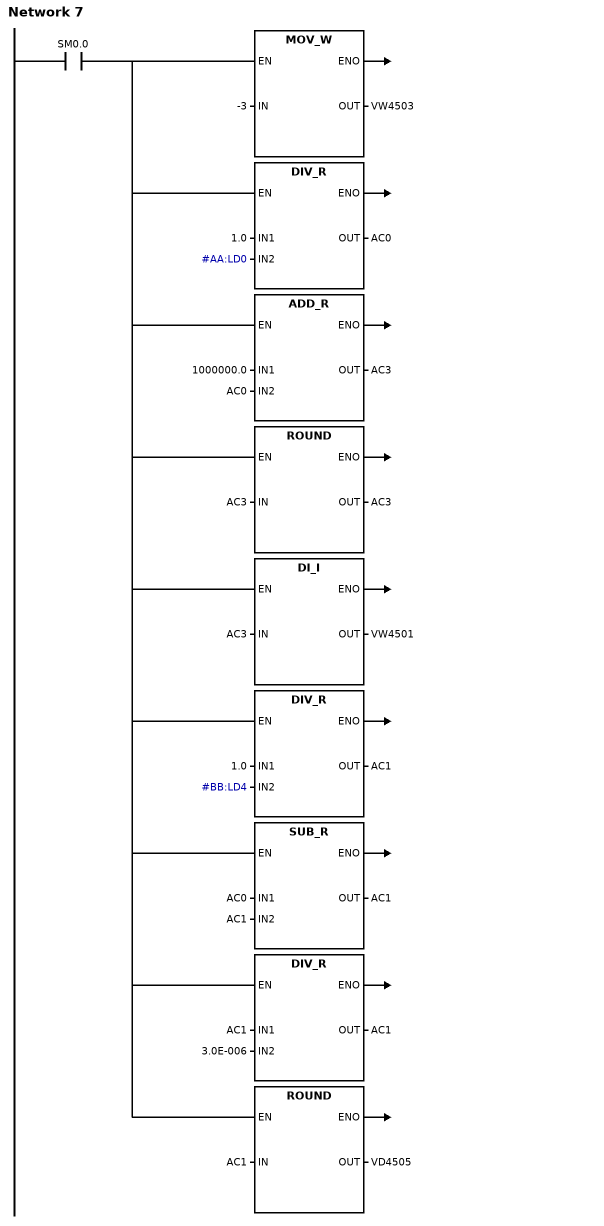
[picture p24: SBR5 networks 7-7]
Network 7
LD     SM0.0
MOVW   -3, VW4503
MOVR   1.0, AC0
/R     #AA:LD0, AC0
MOVR   1000000.0, AC3
+R     AC0, AC3
ROUND  AC3, AC3
DTI    AC3, VW4501
MOVR   1.0, AC1
/R     #BB:LD4, AC1
*R     -1.0, AC1
+R     AC0, AC1
/R     3.0E-006, AC1
ROUND  AC1, VD4505
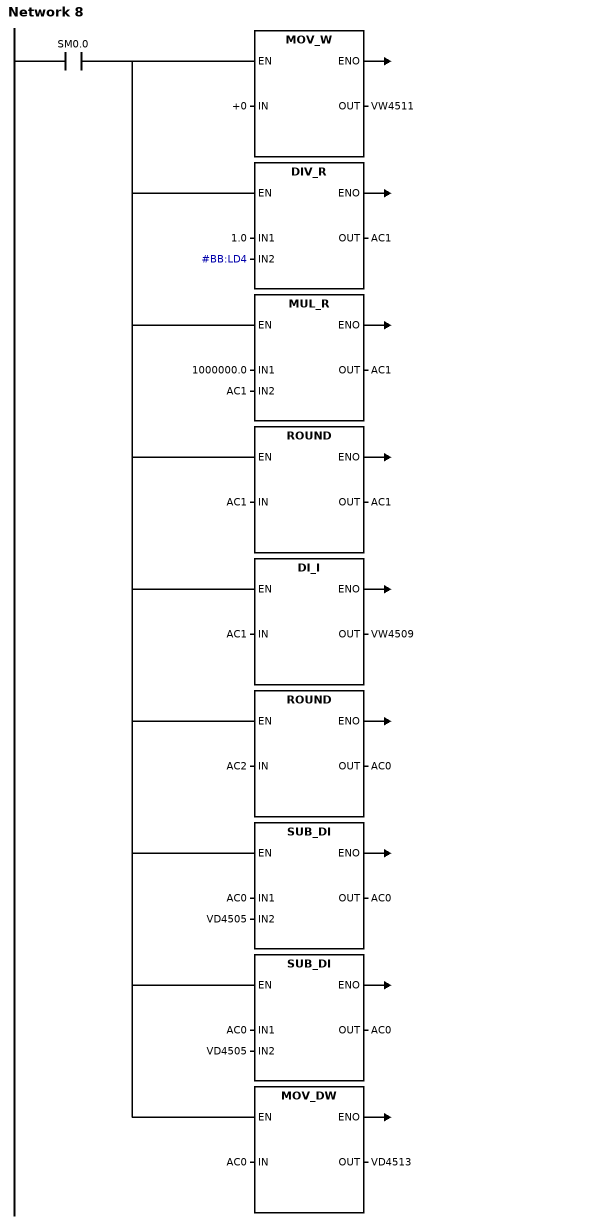
Network 8
LD     SM0.0
MOVW   +0, VW4511
MOVR   1.0, AC1
/R     #BB:LD4, AC1
*R     1000000.0, AC1
ROUND  AC1, AC1
DTI    AC1, VW4509
ROUND  AC2, AC0
-D     VD4505, AC0
-D     VD4505, AC0
MOVD   AC0, VD4513
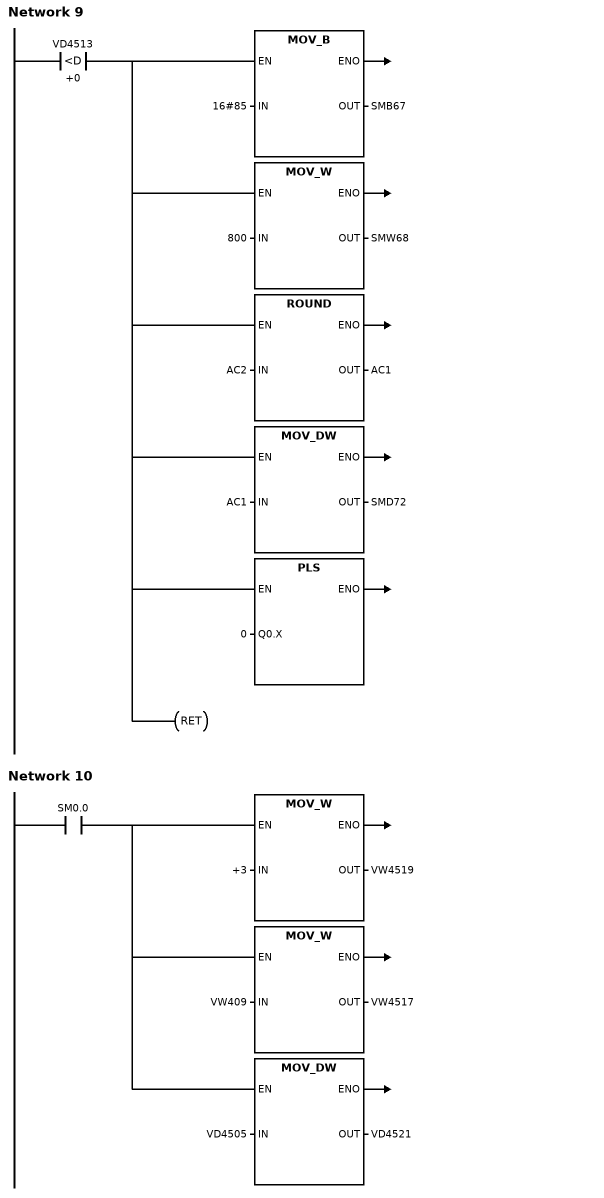
Network 9
LDD<   VD4513, +0
MOVB   16#85, SMB67
MOVW   800, SMW68
ROUND  AC2, AC1
MOVD   AC1, SMD72
PLS    0
CRET
Network 10
LD     SM0.0
MOVW   +3, VW4519
MOVW   VW409, VW4517
MOVD   VD4505, VD4521
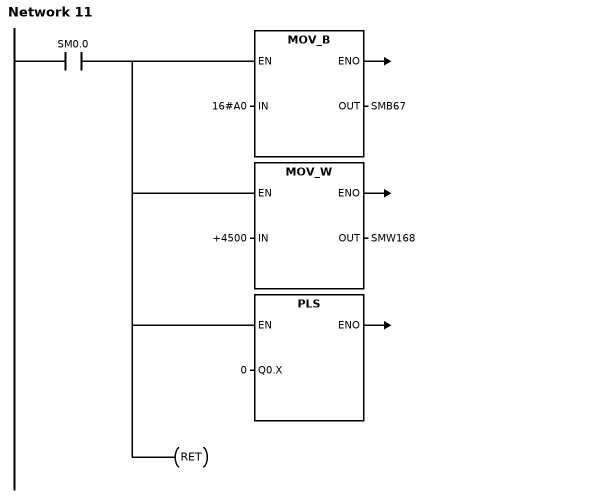
Network 11
LD     SM0.0
MOVB   16#A0, SMB67
MOVW   +4500, SMW168
PLS    0
CRET
END_SUBROUTINE_BLOCK

SUBROUTINE_BLOCK stop_ch0:SBR6
TITLE=stop_ch0
BEGIN
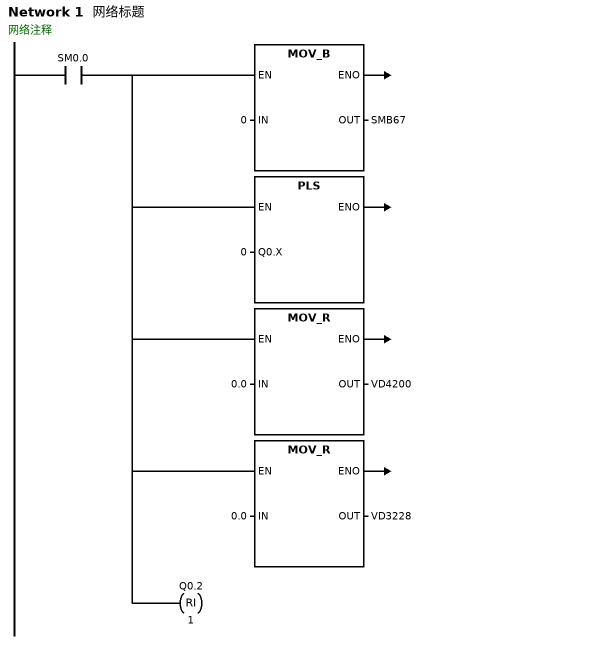
Network 1 // 网络标题
// 网络注释
LD     SM0.0
MOVB   0, SMB67
PLS    0
MOVR   0.0, VD4200
MOVR   0.0, VD3228
RI     Q0.2, 1
END_SUBROUTINE_BLOCK

SUBROUTINE_BLOCK pls_ch1:SBR7
TITLE=子程序7  //脉冲发生器2的控制程序
VAR_INPUT
AA:REAL;	// LD0 
BB:REAL;	// LD4 
CC:REAL;	// LD8 
END_VAR
BEGIN
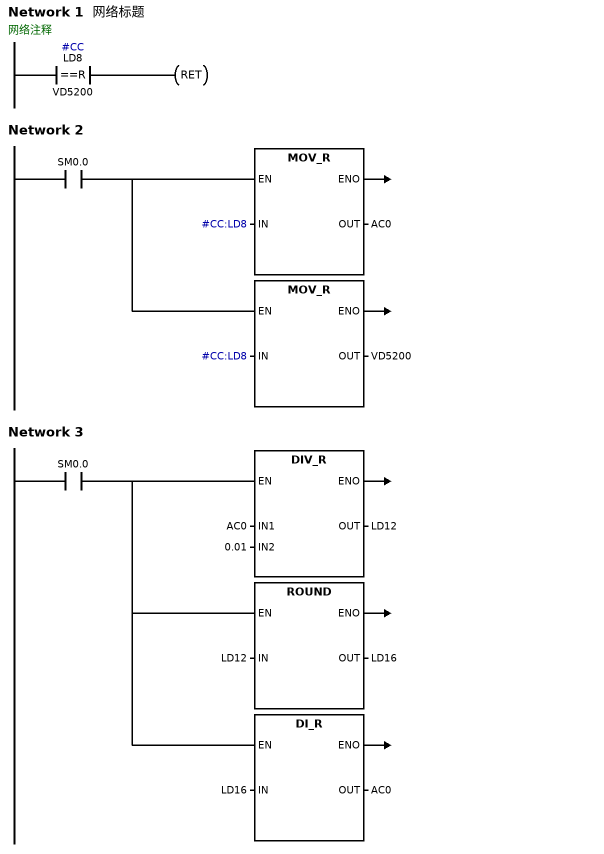
Network 1 // 网络标题
// 网络注释
LDR=   #CC:LD8, VD5200
CRET
Network 2
LD     SM0.0
MOVR   #CC:LD8, AC0
MOVR   #CC:LD8, VD5200
Network 3
LD     SM0.0
MOVR   AC0, LD12
/R     0.01, LD12
ROUND  LD12, LD16
DTR    LD16, AC0
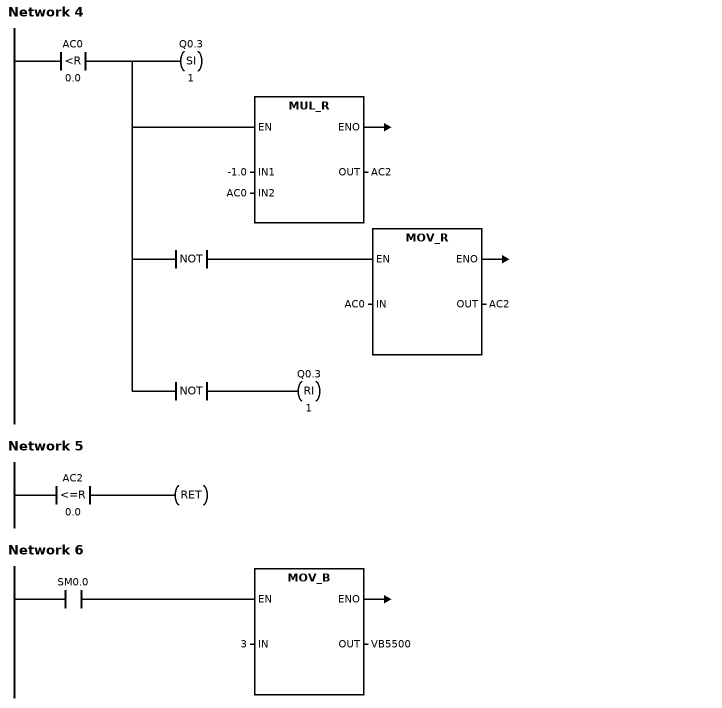
Network 4
LDR<   AC0, 0.0
LPS
SI     Q0.3, 1
MOVR   -1.0, AC2
*R     AC0, AC2
NOT
MOVR   AC0, AC2
LPP
NOT
RI     Q0.3, 1
Network 5
LDR<=  AC2, 0.0
CRET
Network 6
LD     SM0.0
MOVB   3, VB5500
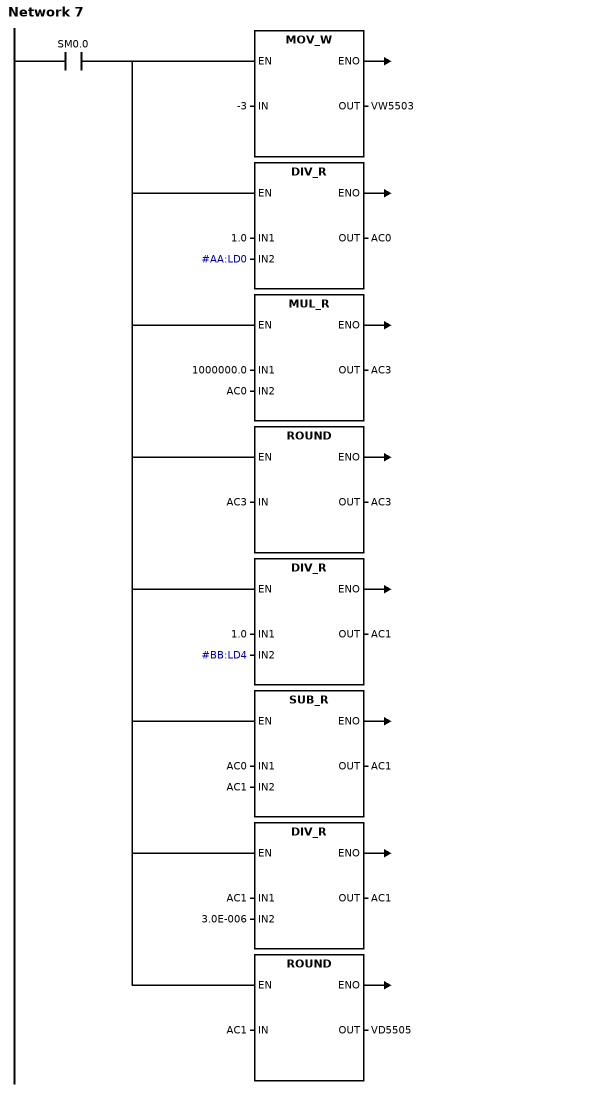
Network 7
LD     SM0.0
MOVW   -3, VW5503
MOVR   1.0, AC0
/R     #AA:LD0, AC0
MOVR   1000000.0, AC3
*R     AC0, AC3
ROUND  AC3, AC3
MOVR   1.0, AC1
/R     #BB:LD4, AC1
*R     -1.0, AC1
+R     AC0, AC1
/R     3.0E-006, AC1
ROUND  AC1, VD5505
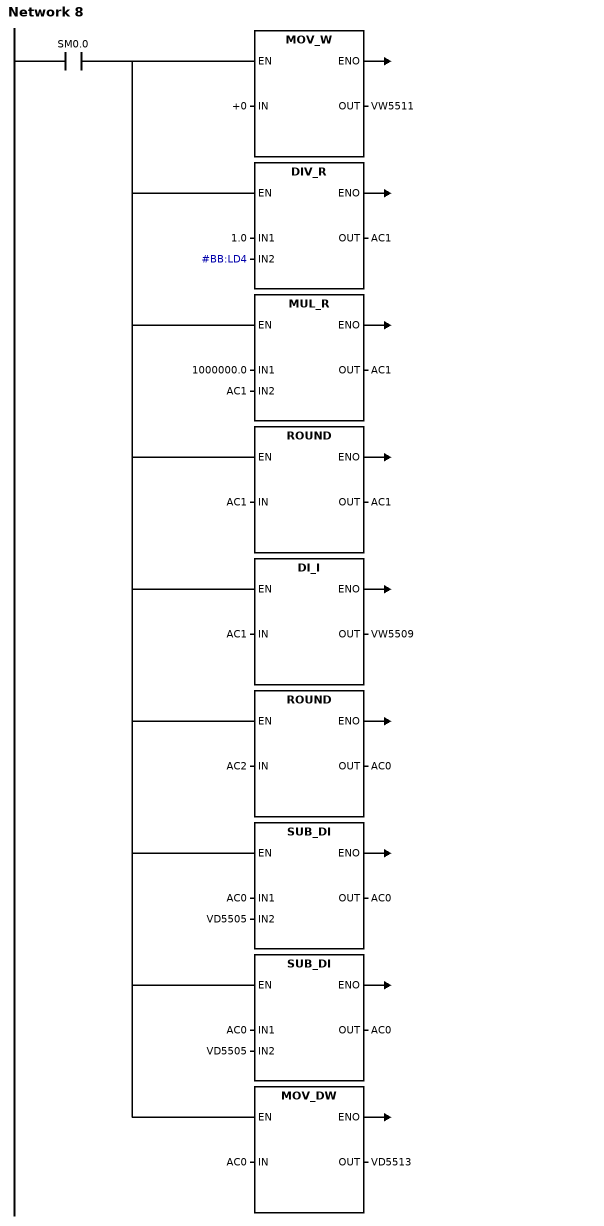
Network 8
LD     SM0.0
MOVW   +0, VW5511
MOVR   1.0, AC1
/R     #BB:LD4, AC1
*R     1000000.0, AC1
ROUND  AC1, AC1
DTI    AC1, VW5509
ROUND  AC2, AC0
-D     VD5505, AC0
-D     VD5505, AC0
MOVD   AC0, VD5513
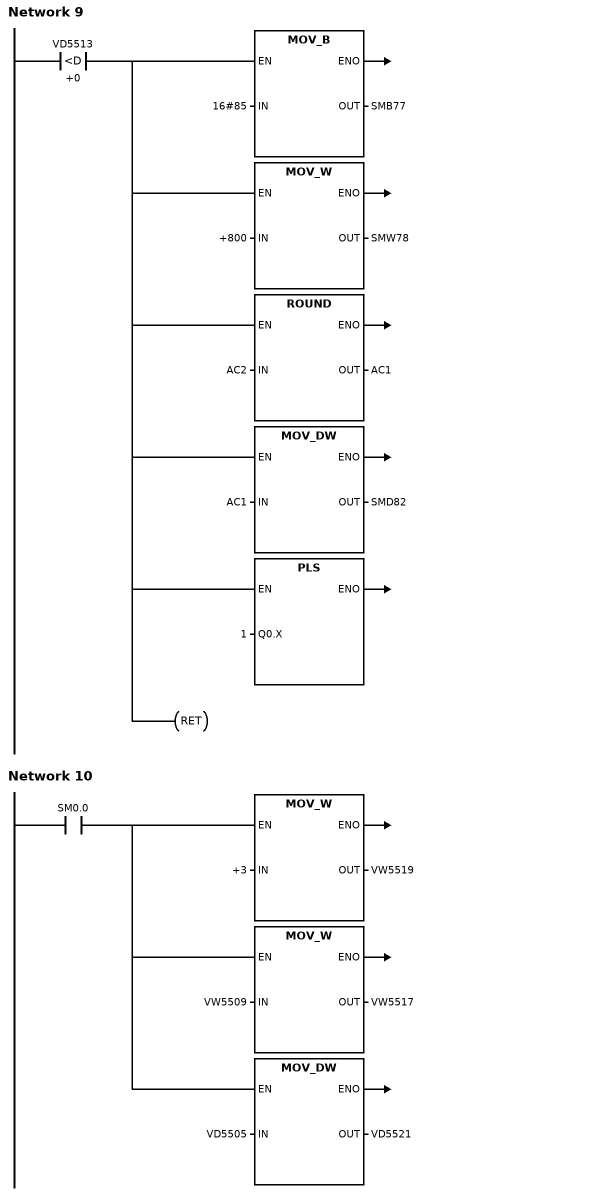
Network 9
LDD<   VD5513, +0
MOVB   16#85, SMB77
MOVW   +800, SMW78
ROUND  AC2, AC1
MOVD   AC1, SMD82
PLS    1
CRET
Network 10
LD     SM0.0
MOVW   +3, VW5519
MOVW   VW5509, VW5517
MOVD   VD5505, VD5521
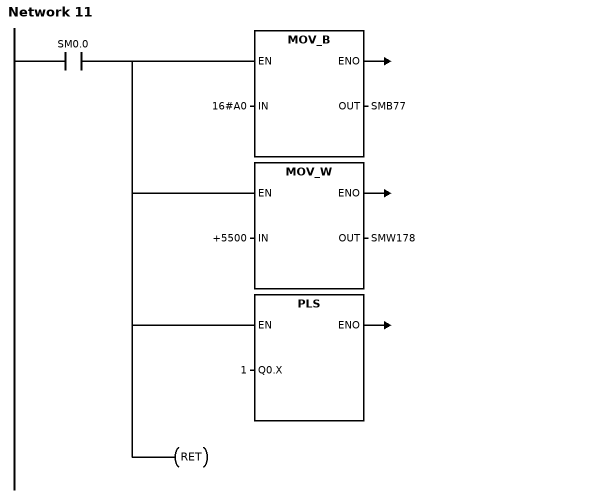
Network 11
LD     SM0.0
MOVB   16#A0, SMB77
MOVW   +5500, SMW178
PLS    1
CRET
END_SUBROUTINE_BLOCK

SUBROUTINE_BLOCK stop_ch1:SBR8
TITLE=stop_ch1
BEGIN
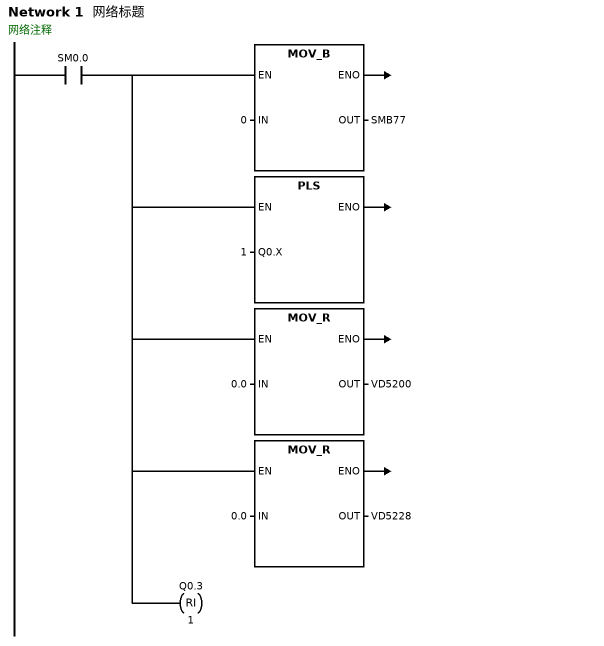
Network 1 // 网络标题
// 网络注释
LD     SM0.0
MOVB   0, SMB77
PLS    1
MOVR   0.0, VD5200
MOVR   0.0, VD5228
RI     Q0.3, 1
END_SUBROUTINE_BLOCK

DATA_BLOCK_TAB 用户定义1
BEGIN
//数据页注释
//按 F1 键获取帮助和示范数据页
//仓库x轴坐标值
VD616    10
VD620    97
VD624    184
VD628    271
//仓库y轴坐标值
VD600    7.9
VD604    94.9
VD608    181.9
VD612    268.9
END_DATA_BLOCK_TAB
